PROGRAM MAIN
VAR
	temperatureSimul:FB_Process;
	tempCmd AT %I*:LREAL;
	actualTemp AT %Q*:LREAL;
END_VAR
VAR CONSTANT
	taskCycletime:TIME:=T#10MS;
	bNoiseEnable:BOOL:=TRUE;
END_VAR

temperatureSimul(fY:= tempCmd, tTa:=taskCycletime , bNoise:= bNoiseEnable, fX=>actualTemp);

END_PROGRAM

(* stored: Version 1.1.0.1, ProductVersion 3.1.4024.12
   POU MAIN: Id {802f900f-cdd4-480e-acdf-5193ea5f97a2}, SpecialFunc None *)
